// TIA Portal project "BloqueFuncionFB" (V16)

(* hardware
DEVICE "S7-1200 station_1"  S7-1200 Station
   slot 0: "Rack_0"  S7-1200 Rack  Rack  V1.0
   slot 1: "PLC_1"  CPU 1214C AC/DC/Rly  6ES7 214-1BG40-0XB0  V4.4
*)

// ===== PLC "PLC_1"  CPU 1214C AC/DC/Rly =====

VAR_GLOBAL   // PLC tag table "Tabla de variables estándar"
   "Tag_1" AT %I1.0 : Bool;
   "Tag_2" AT %I1.1 : Bool;
   "Tag_3" AT %Q1.0 : Bool;
   "Tag_4" AT %I1.2 : Bool;
   "Tag_5" AT %I1.3 : Bool;
   "Tag_6" AT %Q1.1 : Bool;
   "Tag_7" AT %I1.4 : Bool;
   "Tag_8" AT %I1.5 : Bool;
   "Tag_9" AT %Q1.2 : Bool;
END_VAR

DATA_BLOCK "motor1"   // DB1
{ S7_Optimized_Access := 'TRUE' }
VERSION : 0.1
// stored: InstanceOfName Bloque_1
"Bloque_1"
BEGIN
END_DATA_BLOCK

DATA_BLOCK "motor2"   // DB2
{ S7_Optimized_Access := 'TRUE' }
VERSION : 0.1
// stored: InstanceOfName Bloque_1
"Bloque_1"
BEGIN
END_DATA_BLOCK

DATA_BLOCK "motor3"   // DB3
{ S7_Optimized_Access := 'TRUE' }
VERSION : 0.1
// stored: InstanceOfName Bloque_1
"Bloque_1"
BEGIN
END_DATA_BLOCK

FUNCTION_BLOCK "Bloque_1"   // FB1, LAD
{ S7_Optimized_Access := 'TRUE' }
VERSION : 0.1
// Arranque temporizado de motores. Se agrega parada de motor con salida de ton y con pulsador stop.
   VAR_INPUT
      START : Bool;
      STOP : Bool;
      TIEMPO : Time;
   END_VAR
   VAR_OUTPUT
      MOTOR : Bool;
   END_VAR
   VAR
      IEC_Timer_0_Instance : TON_TIME;
   END_VAR
   VAR_TEMP   // added for the SCL form of the ladder/FBD networks
      _w1 : Bool;
   END_VAR
BEGIN

REGION Network 1
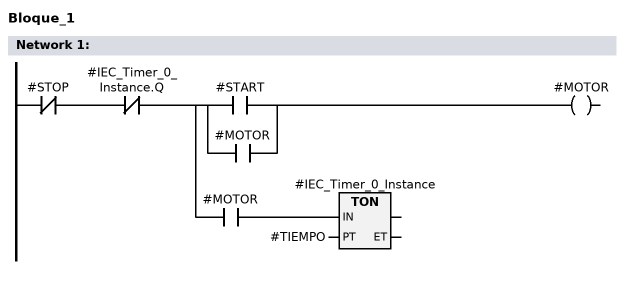
   #_w1 := NOT #STOP AND NOT #IEC_Timer_0_Instance.Q;
   #MOTOR := #_w1 AND (#START OR #MOTOR);
   #IEC_Timer_0_Instance(IN := #_w1 AND #MOTOR, PT := #TIEMPO);   // TON
END_REGION
END_FUNCTION_BLOCK

ORGANIZATION_BLOCK "Main"   // OB1, LAD, ProgramCycle
TITLE = "Main Program Sweep (Cycle)"
{ S7_Optimized_Access := 'TRUE' }
VERSION : 0.1
   VAR_INPUT
      Initial_Call : Bool;   // Initial call of this OB
      Remanence : Bool;   // =True, if remanent data are available
   END_VAR
BEGIN

REGION Network 1
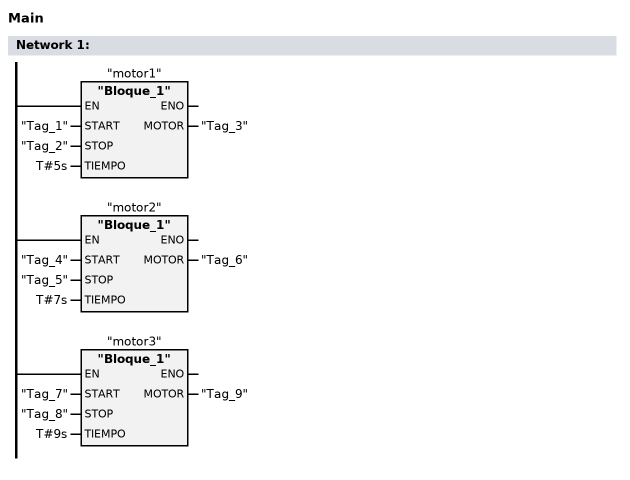
   RUNG wire#powerrail
      "motor1"(START := "Tag_1", STOP := "Tag_2", TIEMPO := T#5s, MOTOR => "Tag_3")
   END_RUNG
   RUNG wire#powerrail
      "motor2"(START := "Tag_4", STOP := "Tag_5", TIEMPO := T#7s, MOTOR => "Tag_6")
   END_RUNG
   RUNG wire#powerrail
      "motor3"(START := "Tag_7", STOP := "Tag_8", TIEMPO := T#9s, MOTOR => "Tag_9")
   END_RUNG
   // the same network as SCL:
   "motor1"(START := "Tag_1", STOP := "Tag_2", TIEMPO := T#5s, MOTOR => "Tag_3");   // "Bloque_1"
   "motor2"(START := "Tag_4", STOP := "Tag_5", TIEMPO := T#7s, MOTOR => "Tag_6");   // "Bloque_1"
   "motor3"(START := "Tag_7", STOP := "Tag_8", TIEMPO := T#9s, MOTOR => "Tag_9");   // "Bloque_1"
END_REGION
END_ORGANIZATION_BLOCK